// TwinCAT 3 PLC project Untitled1
// ProgramVersion: 3.1.4024.0
// libraries:
//   Tc2_Standard, * (Beckhoff Automation GmbH)
//   Tc2_System, * (Beckhoff Automation GmbH)
//   Tc3_Module, * (Beckhoff Automation GmbH)
// project tree:
//   / GlobalTextList.TcGTLO, PlcTask.TcTTO (not stored), Visualization Manager.TcVMO (not stored)
//   GVLs/ GIOL.TcGVL, Global_IO_assignment.TcPOU (not stored), GVL.TcGVL (not stored)
//   POUs/ BINARY_TO_DEC.TcPOU (not stored), BLINK.TcPOU, LIFT.TcPOU, MAIN.TcPOU, INMODE.TcPOU (not stored), Pulse.TcPOU (not stored), ROBOT_BIT_TRL.TcPOU (not stored)
//   VISUs/ StandardPLCversenyVISU.TcVIS
// real-time tasks:
//   TASK PlcTask: cycle T#10ms, priority 20, ADS port 350
// I/O:
//   DEVICE Device 1 (EtherCAT), AmsNetId 26.197.133.186.2.1
//     Term 1 (EK1200) [EK1200-5000 EtherCAT Power supply (2A E-Bus)]
//       Term 2 (EL1008) [EL1008 8Ch. Dig. Input 24V, 3ms]
//       Term 3 (EL1008) [EL1008 8Ch. Dig. Input 24V, 3ms]
//       Term 4 (EL2008) [EL2008 8Ch. Dig. Output 24V, 0.5A]
//       Term 5 (EL2008) [EL2008 8Ch. Dig. Output 24V, 0.5A]
//       Term 6 (EL9011) [EL9011 End Terminal]
// variable links:
//   Untitled1/Untitled1 Instance <-> Device 1 (EtherCAT)/Term 1 (EK1200)/Term 2 (EL1008)
//     PlcTask Inputs/GIOL.xIn{0..7} <-> Channel {1..8}/Input  (8 links)
//   Untitled1/Untitled1 Instance <-> Device 1 (EtherCAT)/Term 1 (EK1200)/Term 3 (EL1008)
//     PlcTask Inputs/GIOL.xIn{8..15} <-> Channel {1..8}/Input  (8 links)
//   Untitled1/Untitled1 Instance <-> Device 1 (EtherCAT)/Term 1 (EK1200)/Term 4 (EL2008)
//     PlcTask Outputs/GIOL.Out{0..7} <-> Channel {1..8}/Output  (8 links)
//   Untitled1/Untitled1 Instance <-> Device 1 (EtherCAT)/Term 1 (EK1200)/Term 5 (EL2008)
//     PlcTask Outputs/GIOL.Out{8..15} <-> Channel {1..8}/Output  (8 links)

// ---- GVLs/GIOL.TcGVL
{attribute 'qualified_only'}
VAR_GLOBAL
	xIn0 	AT%IX0.0:	BOOL;
	xIn1 	AT%IX0.1:	BOOL;
	xIn2 	AT%IX0.2:	BOOL;
	xIn3 	AT%IX0.3:	BOOL;
	xIn4 	AT%IX0.4:	BOOL;
	xIn5 	AT%IX0.5:	BOOL;
	xIn6 	AT%IX0.6:	BOOL;
	xIn7 	AT%IX0.7:	BOOL;
	
	xIn8 	AT%IX1.0:	BOOL;
	xIn9 	AT%IX1.1:	BOOL;
	xIn10 	AT%IX1.2:	BOOL;
	xIn11 	AT%IX1.3:	BOOL;
	xIn12 	AT%IX1.4:	BOOL;
	xIn13 	AT%IX1.5:	BOOL;
	xIn14 	AT%IX1.6:	BOOL;
	xIn15 	AT%IX1.7:	BOOL;
	
	Out0 	AT%QX0.0:	BOOL;
	Out1 	AT%QX0.1:	BOOL;
	Out2 	AT%QX0.2:	BOOL;
	Out3 	AT%QX0.3:	BOOL;
	Out4 	AT%QX0.4:	BOOL;
	Out5 	AT%QX0.5:	BOOL;
	Out6 	AT%QX0.6:	BOOL;
	Out7 	AT%QX0.7:	BOOL;
	
	
	Out8 	AT%QX1.0:	BOOL;
	Out9 	AT%QX1.1:	BOOL;
	Out10 	AT%QX1.2:	BOOL;
	Out11 	AT%QX1.3:	BOOL;
	Out12 	AT%QX1.4:	BOOL;
	Out13 	AT%QX1.5:	BOOL;
	Out14 	AT%QX1.6:	BOOL;
	Out15 	AT%QX1.7:	BOOL;
	
	In0 	:	BOOL;
	In1 	:	BOOL;
	In2 	:	BOOL;
	In3 	:	BOOL;
	In4 	:	BOOL;
	In5 	:	BOOL;
	In6 	:	BOOL;
	In7 	:	BOOL;
	
	In8 	:	BOOL;
	In9 	:	BOOL;
	In10 	:	BOOL;
	In11 	:	BOOL;
	In12 	:	BOOL;
	In13 	:	BOOL;
	In14 	:	BOOL;
	In15 	:	BOOL;
	
	bIn0 	:	BOOL;
	bIn1 	:	BOOL;
	bIn2 	:	BOOL;
	bIn3 	:	BOOL;
	bIn4 	:	BOOL;
	bIn5 	:	BOOL;
	bIn6 	:	BOOL;
	bIn7 	:	BOOL;
	
	bIn8 	:	BOOL;
	bIn9 	:	BOOL;
	bIn10 	:	BOOL;
	bIn11 	:	BOOL;
	bIn12 	:	BOOL;
	bIn13 	:	BOOL;
	bIn14 	:	BOOL;
	bIn15 	:	BOOL;
	
	TaskName : WSTRING := "Null Task";
	CaseNum  : INT := 0;
	
	TaskName2 : WSTRING := "Null Task";
	CaseNum2 : INT := 0;
	
END_VAR

// ---- POUs/BLINK.TcPOU
FUNCTION_BLOCK BLINK
VAR_INPUT
	TOGGLE : BOOL; // Indítja és leállítja a villogást
	ON_TIME : TIME; // Bekapcsolva töltött idő
	OFF_TIME : TIME; // Kikapcsolva töltött idő
END_VAR
VAR_OUTPUT
	LED : BOOL; // A led változó ami villogni fog
END_VAR
VAR
	clk1 :TON;
	clk2 :TON;
	i: INT;
END_VAR

clk1(PT:=ON_TIME);
clk2(PT:=OFF_TIME);
IF TOGGLE  THEN
	CASE i OF

0:
LED := TRUE;
clk1.IN := TRUE;
clk2.IN := FALSE;
IF clk1.Q THEN
i :=1;  
END_IF
1:
LED := FALSE;
clk1.IN := FALSE;
clk2.IN := TRUE;
IF clk2.Q THEN
	i := 0;
END_IF
	END_CASE
ELSE
		LED := FALSE;
		i:=0;
END_IF

END_FUNCTION_BLOCK

// ---- POUs/LIFT.TcPOU
FUNCTION_BLOCK LIFT
VAR_INPUT
	LiftRun : BOOL;
	DOOR_OPEN : BOOL;    //
	RaklapInLift : BOOL; // I 0.6
	
	
	//PalettLoaded : BOOL;
END_VAR
VAR_OUTPUT
	LiftUp : BOOL;
	LiftDown : BOOL;
	LiftEnd : BOOL;
	LiftReady : BOOL;
	LiftPos : INT;	
	Raklap_IN : BOOL; //Raklap be szalag 
	Raklap_OUT :BOOL; //Raklap ki szalag
	Raklap_MID : BOOL;
	
END_VAR



VAR
CaseN : INT;	
F_Ready : F_TRIG;
LayerCount : INT;
Open_TIME : TON;
PUSH_OUT : TON;
Rtrig : R_TRIG;

END_VAR





PUSH_OUT(IN:= Raklap_OUT, PT := T#3S);


Open_TIME(IN:=DOOR_OPEN, PT:= T#4S);

Rtrig(CLK:=Open_TIME.Q);


IF Rtrig.Q THEN
	
	LayerCount := LayerCount + 1;
END_IF


CASE CaseN OF

	
0:
		Raklap_IN := 1;
		Raklap_MID := 1;
		
	IF RaklapInLift THEN 
	Raklap_IN := 0;   // Raklap bent
	Raklap_MID := 0;
		CaseN := 20;
	
	END_IF
20:							//lift felmegy
		LiftUp := 1;
		LiftEnd := 1;
		LayerCount := 0;   //Layer reset
	IF LiftRun = 0 THEN
		CaseN := 30;
		LiftPos := 0;
		
	
	END_IF
30:						//Lift lemegy egy lépést
	LiftDown:= 1;
	CaseN:= 31;
	LiftUp := 0;
	LiftEnd := 0;
	
	
31:
LiftDown := 0;
IF LiftRun = 0 THEN
LiftReady := 1;
LiftPos := 1;
CaseN := 40;
END_IF


40:
	
IF LayerCount = 1 THEN   // első sor megvan le mozog a lift
	LiftDown := 1;
	LiftReady := 0;
	
	CaseN := 41;
	END_IF
41:
LiftDown := 0;
IF LiftRun = 0 THEN     
LiftReady := 1;
LiftPos := 2;
CaseN := 40;
END_IF


50: 

IF LayerCount = 2 THEN   // második sor megvan le mozog a lift
	LiftDown := 1;
	LiftReady := 0;
	
	CaseN := 51;
	END_IF
51:
LiftDown := 0;
IF LiftRun = 0 THEN     
LiftReady := 1;
LiftPos := 3;
CaseN := 60;
END_IF

60: 

IF LayerCount = 2 THEN   // Harmadik sor megvan le mozog a lift végállásig
	LiftDown := 1;
	LiftEnd := 1;
	LiftReady := 0;
	
	CaseN := 61;
	END_IF
61:

IF LiftRun = 0 THEN      
LiftPos := 4;
LiftDown := 0;
LiftEnd := 0;
CaseN := 70;
END_IF
	
70:										//Lift kirakod
	Raklap_OUT := 1;
	Raklap_MID := 1;
	CaseN := 71;
	
71:
	IF PUSH_OUT.Q = 1 THEN
		Raklap_OUT := 0;
		Raklap_MID := 0;
		CaseN := 0;
	END_IF


END_CASE

END_FUNCTION_BLOCK

// ---- POUs/MAIN.TcPOU
PROGRAM MAIN
VAR
	INMODE : INMODE;
	
	Timer : TON;
	TimerT : TIME;
	TimerSW : BOOL;
	
	FallTrig : F_TRIG;
	FallTrigCLK : BOOL;
	
	RiseTrig : R_TRIG;
	RiseTrigCLK : BOOL;
	
	Pulse : Pulse;
	PulseSIGNAL : BOOL; 
	PulseTime : TIME;
	
	N1: INT:=555;
	N2: INT;
	Task : WSTRING;
	Task2: WSTRING;
	Logs : WSTRING;
	
	Carry_IN : BOOL;
	Press : BOOL;
	Track_IN : BOOL;
	Alert_1 : BOOL;
	Lift_UP : BOOL;
	Lift_DOWN : BOOL;
	Lift_END : BOOL;
	Lift_IN  : BOOL;
	Palett_IN : BOOL;
	Palett_GRAB : BOOL;
	Palett_PUSH : BOOL;
	Flap : BOOL;
	Palett_OPEN : BOOL;
	Track_OUT : BOOL;
	Horn : BOOL;
	Alert_2 : BOOL;
	
	Carry_IN_FULL : BOOL;
	Press_FULL : BOOL;
	Press_END : BOOL;
	System_OK : BOOL;
	Track_IN_EMPTY : BOOL;
	Track_OUT_EMPTY : BOOL;
	Lift_FRONT : BOOL;
	Lift_BACK : BOOL;
	Lift_RUN : BOOL;
	Palett_PUSH_END : BOOL;
	Palett_CLOSED : BOOL;
	Palett_GRAB_OK : BOOL;
	Auto_SWITCH : BOOL;
	START : BOOL;
	STOP : BOOL;
	RESET : BOOL;
	
	BOX_Count : INT := 0;
	Line_Count : INT := 0;
	Layer_Count : INT := 0;
	RAK_Count : INT := 0;
	
	Stack_MODE : BOOL := TRUE; //if 1 then 3x2; if 0 then 2x3
	Layer_READY : BOOL;
	
	BOX_Count_FULL : BOOL;
	Line_Count_FULL : BOOL;
	Lift_OK : BOOL;
	
	
	LIFT : LIFT;
	
END_VAR

INMODE(); 
GIOL.TaskName := Task;
GIOL.CaseNum := N1;

GIOL.TaskName2 := Task2;
GIOL.CaseNum2 := N2;

Carry_IN_FULL := GIOL.In0;
Press_FULL := GIOL.In1;
Press_END := GIOL.In2;
System_OK := GIOL.In3;
Track_IN_EMPTY := GIOL.In4;
Track_OUT_EMPTY := GIOL.In5;
Lift_FRONT := GIOL.In6;
Lift_BACK := GIOL.In7;
Lift_RUN := GIOL.In8;
Palett_PUSH_END := GIOL.In9;
Palett_CLOSED := GIOL.In10;
Palett_GRAB_OK := GIOL.In11;
Auto_SWITCH := GIOL.In12;
START := GIOL.In13;
STOP := GIOL.In14;
RESET := GIOL.In15;

GIOL.Out0 := Carry_IN;
GIOL.Out1 := Press;
GIOL.Out2 := Track_IN;
GIOL.Out3 := Alert_1;
GIOL.Out4 := Lift_UP;
GIOL.Out5 := Lift_DOWN;
GIOL.Out6 := Lift_END;
GIOL.Out7 := Lift_IN;
GIOL.Out8 := Palett_PUSH;
GIOL.Out9 := Palett_GRAB;
GIOL.Out10 := Palett_IN;
GIOL.Out11 := Flap;
GIOL.Out12 := Palett_OPEN;
GIOL.Out13 := Track_OUT;
GIOL.Out14 := Horn;
GIOL.Out15 := Alert_2;

IF System_OK THEN 

IF NOT(N1 = 555 OR N1= 666) THEN
	LIFT(LiftRun:=Lift_RUN,DOOR_OPEN:=Palett_OPEN ,RaklapInLift:=Lift_FRONT);
	Lift_UP := LIFT.LiftUp;
	Lift_DOWN := LIFT.LiftDown;
	Lift_END := LIFT.LiftEnd;
	Lift_OK := LIFT.LiftReady;
	Track_IN := LIFT.Raklap_IN;
	Track_OUT := LIFT.Raklap_OUT;
	Timer(IN:=TimerSW,PT:=TimerT);
	FallTrig(CLK:=FallTrigCLK);
	RiseTrig(CLK:=Carry_IN_FULL);
	Pulse(SIGNAL:=PulseSIGNAL,Pulse_time:=PulseTime);
	Lift_IN := LIFT.Raklap_MID;
END_IF



//STACK MODE
IF Stack_MODE THEN
	Flap:=FALSE;
	IF Line_Count = 3 THEN
			Line_Count := 0;
			Line_Count_FULL :=TRUE;
			Layer_Count := Layer_Count +1;
	END_IF
	IF BOX_Count = 3 THEN
		BOX_Count := 1;
		BOX_Count_FULL := TRUE;
	END_IF
ELSE
	Flap:=TRUE;
	IF Line_Count = 2 THEN
			Line_Count := 0;
			Line_Count_FULL :=TRUE;
			Layer_Count := Layer_Count +1;
	END_IF
	IF BOX_Count = 4 THEN
		BOX_Count := 0;
		BOX_Count_FULL := TRUE;
	END_IF
	
END_IF

IF Layer_Count = 3 THEN
	Layer_Count := 0;
	Stack_MODE  := NOT Stack_MODE;
END_IF

// PRESS {
IF Press THEN
	Press:=FALSE;
END_IF

IF Press_FULL AND Press_END THEN
	Press:=TRUE;
END_IF
//} Press

IF RiseTrig.Q THEN
	BOX_Count := BOX_Count + 1;
END_IF

//Async TASK_1 { Carry_IN, Palett_ALL
//

IF RESET THEN
	Carry_IN := FALSE;
	Press := FALSE;
	Track_IN := FALSE;
	Alert_1 := FALSE;
	Lift_UP := FALSE;
	Lift_DOWN := FALSE;
	Lift_END := FALSE;
	Lift_IN  := FALSE;
	Palett_IN := FALSE;
	Palett_GRAB := FALSE;
	Palett_PUSH := FALSE;
	Flap := FALSE;
	Palett_OPEN := FALSE;
	Track_OUT := FALSE;
	Horn := FALSE;
	Alert_2 := FALSE;
	
	BOX_Count := 0;
	Line_Count := 0;
	Layer_Count := 0;
	RAK_Count := 0;
	
	Stack_MODE := TRUE; //if 1 then 3x2; if 0 then 2x3
	Layer_READY := FALSE;
	
	BOX_Count_FULL := FALSE;
	Line_Count_FULL := FALSE;
	N1:=555;
END_IF

	
CASE N1 OF
	555:Task:="Wait for Auto switch";
		IF Auto_SWITCH THEN
			N1:=666;
		END_IF
		
	666:Task:="Wait for start";
		IF START  THEN
			N1:=0;
		END_IF
	
	0:Task:="Building line";
		Carry_IN := TRUE;
		Palett_IN := TRUE;
		Palett_OPEN := FALSE;
		N1:=10;
		
	10:Task:="Building line";	
		IF BOX_Count_FULL THEN
			Carry_IN := FALSE;
			Palett_IN := FALSE;
			Palett_PUSH := TRUE;
			BOX_Count :=1;
			TimerT:=T#3500MS;
			BOX_Count_FULL := FALSE;
			N1:=20;
		END_IF
		
	20:Task:="Stop Boxes and push line";
		TimerSW:=TRUE;
		IF Timer.Q THEN
			Line_Count := Line_Count + 1;
			TimerSW := FALSE;
			Palett_PUSH := FALSE;
			N1:=30;
		END_IF
		
	30:Task:="Stop Boxes and push line";
		TimerSW := TRUE;
		IF Timer.Q THEN
			TimerSW:=FALSE;
			N1:= 0;
		END_IF
		IF Line_Count_FULL THEN
			N1:=60;
			Line_Count_FULL := FALSE;
			Palett_GRAB := TRUE;
		END_IF
		
	60:Task:="";
		IF Palett_GRAB_OK AND Lift_OK THEN
			Palett_OPEN:=TRUE;
			TimerT:=T#3S;
			N1:=70;
		END_IF
		
	70:Task:="";
		TimerSW:=TRUE;
		IF Timer.Q THEN
			Palett_GRAB := FALSE;
			TimerSW:=FALSE;
			;
		END_IF
	ELSE
		N1:=0;
END_CASE
ELSE
	Carry_IN := FALSE;
	Press := FALSE;
	Track_IN := FALSE;
	Alert_1 := FALSE;
	Lift_UP := FALSE;
	Lift_DOWN := FALSE;
	Lift_END := FALSE;
	Lift_IN  := FALSE;
	Palett_IN := FALSE;
	Palett_GRAB := FALSE;
	Palett_PUSH := FALSE;
	Flap := FALSE;
	Palett_OPEN := FALSE;
	Track_OUT := FALSE;
	Horn := FALSE;
	Alert_2 := FALSE;
	
	BOX_Count := 0;
	Line_Count := 0;
	Layer_Count := 0;
	RAK_Count := 0;
	
	Stack_MODE := TRUE; //if 1 then 3x2; if 0 then 2x3
	Layer_READY := FALSE;
	
	BOX_Count_FULL := FALSE;
	Line_Count_FULL := FALSE;
END_IF

END_PROGRAM

// ---- GlobalTextList.TcGTLO
TEXTLIST GlobalTextList
  169 = ' TrackOUT_EM'
  655 = ' TrackO_EM'
  71 = 'ABCD'
  595 = 'ABCDEFG'
  153 = 'alert'
  855 = 'Alert'
  76 = 'Alert1'
  706 = 'Alert2'
  188 = 'AUTO_SW'
  120 = 'Behszal1'
  920 = 'burn'
  819 = 'CarryIN'
  438 = 'CarryIN_F'
  847 = 'CarryIN_FULL'
  216 = 'CASE: %d'
  900 = 'cir pos1'
  685 = 'cir pos2'
  726 = 'cir pos3'
  672 = 'cirLeft'
  662 = 'cirRight'
  106 = 'Címkéző'
  283 = 'eject'
  404 = 'EXECUTING: %s'
  16 = 'FigyVill1'
  637 = 'Flap'
  947 = 'Görgösm1'
  414 = 'HORN'
  848 = 'IN 0'
  11 = 'IN 1'
  589 = 'inconv'
  929 = 'INPUT MODE'
  57 = 'kem be'
  742 = 'kem in'
  828 = 'kem ki'
  263 = 'kem out'
  441 = 'kem TrackOUT_EM'
  172 = 'kemdoor'
  639 = 'kemfull'
  823 = 'kemfull!'
  463 = 'Life'
  276 = 'LiftBack'
  927 = 'LiftBehLánc'
  334 = 'LiftDOWN'
  998 = 'LiftDW'
  657 = 'LiftEND'
  473 = 'LiftFront'
  841 = 'LiftIN'
  73 = 'LiftUP'
  613 = 'Lift_Run'
  307 = 'man left'
  489 = 'mandown'
  327 = 'manen1'
  743 = 'manen2'
  810 = 'manright'
  207 = 'manvac'
  984 = 'OU 0'
  620 = 'OUT 0'
  877 = 'OUT 1'
  12 = 'PalettGO'
  617 = 'PalettGRAB'
  328 = 'PalettIN'
  158 = 'PalettOPEN'
  719 = 'Palett_GO_E'
  604 = 'PalGO_E'
  292 = 'PalGRAB_OK'
  401 = 'Pal_Closed'
  403 = 'pickupm'
  315 = 'pickupp'
  98 = 'Press'
  238 = 'PressClosed'
  583 = 'PressFULL'
  524 = 'Press_FULL'
  96 = 'read1'
  923 = 'read2'
  519 = 'readtr'
  197 = 'RESET'
  429 = 'robot1'
  515 = 'robot2'
  599 = 'robotin'
  757 = 'robotout'
  696 = 'saw on'
  705 = 'start'
  606 = 'START'
  896 = 'STOP'
  770 = 'systemok'
  840 = 'SystemOK'
  678 = 'Teszt var'
  335 = 'Teszt változó'
  894 = 'Track'
  986 = 'TrackIN'
  129 = 'TrackIN_EM'
  675 = 'TrackIN_EMY'
  903 = 'TrackOUT'
  651 = 'Warning'
END_TEXTLIST

// ---- VISUs/StandardPLCversenyVISU.TcVIS
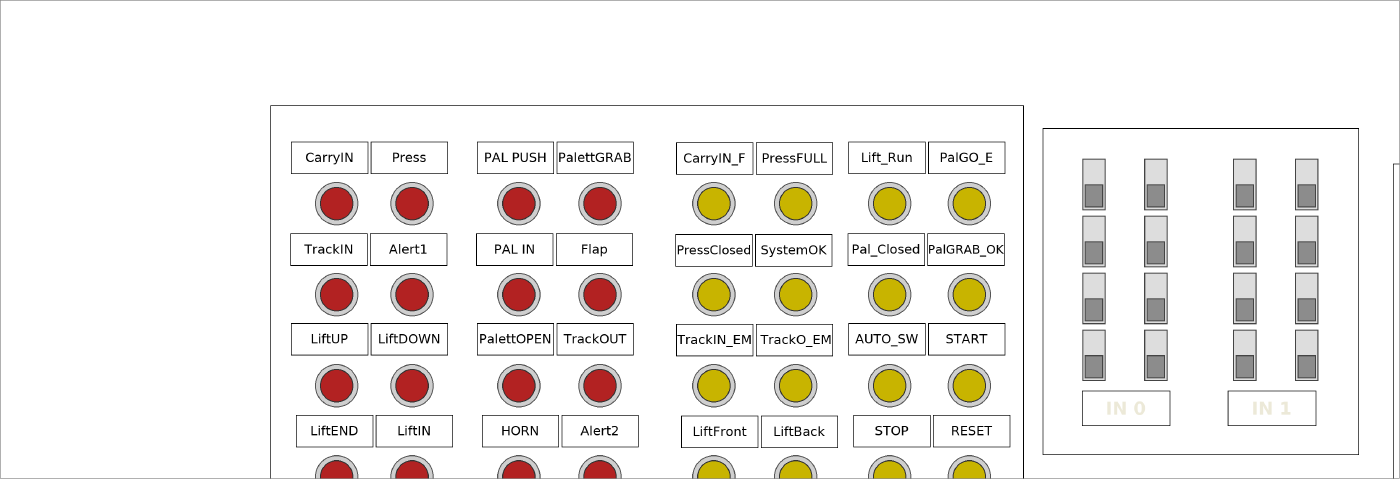
VISUALIZATION StandardPLCversenyVISU  // 1967x673
    Rectangle (1513,674 331x259)
    Rectangle (1957,230 444x459)
    Rectangle (380,148 1058x855)
    Lamp1 (438,251 70x70), variable: GIOL.out0, style: Lamp-Lamp1-Red
    Lamp1 (544,251 70x70), variable: GIOL.out1, style: Lamp-Lamp1-Red
    Lamp1 (694,251 70x70), variable: GIOL.out8, style: Lamp-Lamp1-Red
    Lamp1 (808,251 70x70), variable: GIOL.out9, style: Lamp-Lamp1-Red
    Lamp1 (438,379 70x70), variable: GIOL.out2, style: Lamp-Lamp1-Red
    Lamp1 (544,379 70x70), variable: GIOL.out3, style: Lamp-Lamp1-Red
    Lamp1 (694,379 70x70), variable: GIOL.out10, style: Lamp-Lamp1-Red
    Lamp1 (808,379 70x70), variable: GIOL.out11, style: Lamp-Lamp1-Red
    Lamp1 (438,507 70x70), variable: GIOL.out4, style: Lamp-Lamp1-Red
    Lamp1 (544,507 70x70), variable: GIOL.out5, style: Lamp-Lamp1-Red
    Lamp1 (694,507 70x70), variable: GIOL.out12, style: Lamp-Lamp1-Red
    Lamp1 (808,507 70x70), variable: GIOL.out13, style: Lamp-Lamp1-Red
    Lamp1 (438,635 70x70), variable: GIOL.out6, style: Lamp-Lamp1-Red
    Lamp1 (544,635 70x70), variable: GIOL.out7, style: Lamp-Lamp1-Red
    Lamp1 (694,635 70x70), variable: GIOL.out14, style: Lamp-Lamp1-Red
    Lamp1 (808,635 70x70), variable: GIOL.out15, style: Lamp-Lamp1-Red
    Lamp1 (968,251 70x70), variable: GIOL.in0, style: Lamp-Lamp1-Yellow
    Lamp1 (1083,251 70x70), variable: GIOL.in1, style: Lamp-Lamp1-Yellow
    Lamp1 (1215,251 70x70), variable: GIOL.in8, style: Lamp-Lamp1-Yellow
    Lamp1 (1327,251 70x70), variable: GIOL.in9, style: Lamp-Lamp1-Yellow
    Lamp1 (968,379 70x70), variable: GIOL.in2, style: Lamp-Lamp1-Yellow
    Lamp1 (1083,379 70x70), variable: GIOL.in3, style: Lamp-Lamp1-Yellow
    Lamp1 (1215,379 70x70), variable: GIOL.in10, style: Lamp-Lamp1-Yellow
    Lamp1 (1327,379 70x70), variable: GIOL.in11, style: Lamp-Lamp1-Yellow
    Lamp1 (968,507 70x70), variable: GIOL.in4, style: Lamp-Lamp1-Yellow
    Lamp1 (1083,507 70x70), variable: GIOL.in5, style: Lamp-Lamp1-Yellow
    Lamp1 (1215,507 70x70), variable: GIOL.in12, style: Lamp-Lamp1-Yellow
    Lamp1 (1327,507 70x70), variable: GIOL.in13, style: Lamp-Lamp1-Yellow
    Lamp1 (968,635 70x70), variable: GIOL.in6, style: Lamp-Lamp1-Yellow
    Lamp1 (1083,635 70x70), variable: GIOL.in7, style: Lamp-Lamp1-Yellow
    Lamp1 (1215,635 70x70), variable: GIOL.in14, style: Lamp-Lamp1-Yellow
    Lamp1 (1327,635 70x70), variable: GIOL.in15, style: Lamp-Lamp1-Yellow
    Rectangle (712,722 124x49), "OUT 1"
    Rectangle (1000,714 124x49), "IN 0"
    Rectangle (462,722 124x49), "OUT 0"
    Rectangle (1245,714 124x49), "IN 1"
    Rectangle (497,826 695x68), "EXECUTING: %s", text variable: GIOL.TaskName
    DipSwitch (2077,269 72x80), variable: GIOL.out1, behaviour: TOGGLE, style: Switch-DipSwitch-Gray
    DipSwitch (1990,269 72x80), variable: GIOL.out0, behaviour: TOGGLE, style: Switch-DipSwitch-Gray
    DipSwitch (2077,349 72x80), variable: GIOL.out3, behaviour: TOGGLE, style: Switch-DipSwitch-Gray
    DipSwitch (1990,349 72x80), variable: GIOL.out2, behaviour: TOGGLE, style: Switch-DipSwitch-Gray
    DipSwitch (2077,429 72x80), variable: GIOL.out5, behaviour: TOGGLE, style: Switch-DipSwitch-Gray
    DipSwitch (1990,429 72x80), variable: GIOL.out4, behaviour: TOGGLE, style: Switch-DipSwitch-Gray
    DipSwitch (2077,509 72x80), variable: GIOL.out7, behaviour: TOGGLE, style: Switch-DipSwitch-Gray
    DipSwitch (1990,509 72x80), variable: GIOL.out6, behaviour: TOGGLE, style: Switch-DipSwitch-Gray
    DipSwitch (2289,269 72x80), variable: GIOL.out9, behaviour: TOGGLE, style: Switch-DipSwitch-Gray
    DipSwitch (2202,269 72x80), variable: GIOL.out8, behaviour: TOGGLE, style: Switch-DipSwitch-Gray
    DipSwitch (2289,349 72x80), variable: GIOL.out11, behaviour: TOGGLE, style: Switch-DipSwitch-Gray
    DipSwitch (2202,349 72x80), variable: GIOL.out10, behaviour: TOGGLE, style: Switch-DipSwitch-Gray
    DipSwitch (2289,429 72x80), variable: GIOL.out13, behaviour: TOGGLE, style: Switch-DipSwitch-Gray
    DipSwitch (2202,429 72x80), variable: GIOL.out12, behaviour: TOGGLE, style: Switch-DipSwitch-Gray
    DipSwitch (2289,509 72x80), variable: GIOL.out15, behaviour: TOGGLE, style: Switch-DipSwitch-Gray
    DipSwitch (2202,509 72x80), variable: GIOL.out14, behaviour: TOGGLE, style: Switch-DipSwitch-Gray
    Rectangle (2214,599 124x49), "OUT 1"
    Rectangle (2009,599 124x49), "OUT 0"
    Rectangle (1465,180 444x459)
    DipSwitch (1588,219 72x80), variable: GIOL.bIn1, behaviour: TOGGLE, style: Switch-DipSwitch-Gray
    DipSwitch (1501,219 72x80), variable: GIOL.bIn0, behaviour: TOGGLE, style: Switch-DipSwitch-Gray
    DipSwitch (1588,299 72x80), variable: GIOL.bIn3, behaviour: TOGGLE, style: Switch-DipSwitch-Gray
    DipSwitch (1501,299 72x80), variable: GIOL.bIn2, behaviour: TOGGLE, style: Switch-DipSwitch-Gray
    DipSwitch (1588,379 72x80), variable: GIOL.bIn5, behaviour: TOGGLE, style: Switch-DipSwitch-Gray
    DipSwitch (1501,379 72x80), variable: GIOL.bIn4, behaviour: TOGGLE, style: Switch-DipSwitch-Gray
    DipSwitch (1588,459 72x80), variable: GIOL.bIn7, behaviour: TOGGLE, style: Switch-DipSwitch-Gray
    DipSwitch (1501,459 72x80), variable: GIOL.bIn6, behaviour: TOGGLE, style: Switch-DipSwitch-Gray
    DipSwitch (1800,219 72x80), variable: GIOL.bIn9, behaviour: TOGGLE, style: Switch-DipSwitch-Gray
    DipSwitch (1713,219 72x80), variable: GIOL.bIn8, behaviour: TOGGLE, style: Switch-DipSwitch-Gray
    DipSwitch (1800,299 72x80), variable: GIOL.bIn11, behaviour: TOGGLE, style: Switch-DipSwitch-Gray
    DipSwitch (1713,299 72x80), variable: GIOL.bIn10, behaviour: TOGGLE, style: Switch-DipSwitch-Gray
    DipSwitch (1800,379 72x80), variable: GIOL.bIn13, behaviour: TOGGLE, style: Switch-DipSwitch-Gray
    DipSwitch (1713,379 72x80), variable: GIOL.bIn12, behaviour: TOGGLE, style: Switch-DipSwitch-Gray
    DipSwitch (1800,459 72x80), variable: GIOL.bIn15, behaviour: TOGGLE, style: Switch-DipSwitch-Gray
    DipSwitch (1713,459 72x80), variable: GIOL.bIn14, behaviour: TOGGLE, style: Switch-DipSwitch-Gray
    Rectangle (1725,549 124x49), "IN 1"
    Rectangle (1520,549 124x49), "IN 0"
    Rectangle (1202,826 153x68), "CASE: %d", text variable: GIOL.CaseNum
    DipSwitch (1562,719 116x113), variable: MAIN.INMODE.INState, behaviour: TOGGLE, style: Switch-DipSwitch-Gray
    Rectangle (1572,864 226x49), "INPUT MODE"
    Lamp1 (1707,741 70x70), variable: MAIN.INMODE.INState, style: Lamp-Lamp1-Yellow
    Rectangle (409,199 108x45), "CarryIN"
    Rectangle (521,199 108x45), "Press"
    Rectangle (670,199 108x45), "PAL PUSH"
    Rectangle (782,199 108x45), "PalettGRAB"
    Rectangle (950,200 108x45), "CarryIN_F"
    Rectangle (1062,200 108x45), "PressFULL"
    Rectangle (1192,199 108x45), "Lift_Run"
    Rectangle (1304,199 108x45), "PalGO_E"
    Rectangle (408,328 108x45), "TrackIN"
    Rectangle (520,328 108x45), "Alert1"
    Rectangle (669,328 108x45), "PAL IN"
    Rectangle (781,328 108x45), "Flap"
    Rectangle (949,329 108x45), "PressClosed"
    Rectangle (1061,329 108x45), "SystemOK"
    Rectangle (1191,328 108x45), "Pal_Closed"
    Rectangle (1303,328 108x45), "PalGRAB_OK"
    Rectangle (409,454 108x45), "LiftUP"
    Rectangle (521,454 108x45), "LiftDOWN"
    Rectangle (670,454 108x45), "PalettOPEN"
    Rectangle (782,454 108x45), "TrackOUT"
    Rectangle (950,455 108x45), "TrackIN_EM"
    Rectangle (1062,455 108x45), "TrackO_EM"
    Rectangle (1192,454 108x45), "AUTO_SW"
    Rectangle (1304,454 108x45), "START"
    Rectangle (416,583 108x45), "LiftEND"
    Rectangle (528,583 108x45), "LiftIN"
    Rectangle (677,583 108x45), "HORN"
    Rectangle (789,583 108x45), "Alert2"
    Rectangle (957,584 108x45), "LiftFront"
    Rectangle (1069,584 108x45), "LiftBack"
    Rectangle (1199,583 108x45), "STOP"
    Rectangle (1311,583 108x45), "RESET"
    Rectangle (495,903 695x68), "EXECUTING: %s", text variable: GIOL.TaskName2
    Rectangle (1200,903 153x68), "CASE: %d", text variable: GIOL.CaseNum2
END_VISUALIZATION
